FUNCTION_BLOCK FINAL Receiver IMPLEMENTS I_ReceiverNode, I_Receiver
VAR
	_iCallable		: I_Callable;
	_tag			: Tags.Tag;
	_bIsOk			: BOOL := TRUE;
END_VAR

//FB_Init is always available implicitly and it is used primarily for initialization.
//The return value is not evaluated. For a specific influence, you can also declare the
//methods explicitly and provide additional code there with the standard initialization
//code. You can evaluate the return value.
METHOD FB_Init: BOOL
VAR_INPUT
    bInitRetains: BOOL; // TRUE: the retain variables are initialized (reset warm / reset cold)
    bInCopyCode: BOOL;  // TRUE: the instance will be copied to the copy code afterward (online change)

	iCallable	: I_Callable;
END_VAR
_iCallable := iCallable;
IF _iCallable = 0 THEN
	_bIsOk := FALSE;
	Debug.DebugMsg(THIS^, 'iReceiver = 0!');
END_IF
END_METHOD

PROPERTY INTERNAL IsOk : BOOL
GET
IsOk := _bIsOk;
END_GET
END_PROPERTY

METHOD Pair : Results.Result
VAR_INPUT
	iSignal		: I_Signal;
END_VAR
IF iSignal <> 0 THEN
	Pair := iSignal.Pair(THIS^);
ELSE
	Pair := Results.Error;
END_IF
END_METHOD

METHOD INTERNAL Receive
VAR_INPUT
	iArg			: I_Arg;
END_VAR
_iCallable.Call(iArg);
END_METHOD

PROPERTY Tag : Tags.I_Tag
GET
Tag := _tag;
END_GET
END_PROPERTY

METHOD Unpair : Results.Result
VAR_INPUT
	iSignal		: I_Signal;
END_VAR
IF iSignal <> 0 THEN
	Unpair := iSignal.Unpair(THIS^);
ELSE
	Unpair := Results.Error;
END_IF
END_METHOD

END_FUNCTION_BLOCK

(* stored: Version 1.1.0.1
   POU Receiver: Id {257bc56d-d4ab-4dfa-8333-731f29b2e514}, SpecialFunc None
   Method FB_init: Id {951a002b-ff7a-48cf-b743-6a05c2c3370f}
   Property IsOk: Id {4a36423a-d62a-4434-aa29-147d4a2a72c0}
   Get Get: Id {9181fb34-27f0-4f1d-8d52-cbee4d6fcb65}
   Method Pair: Id {27407187-acff-4901-8f63-f09886ed298e}
   Method Receive: Id {34f6591a-4c68-42fe-83cd-983703da5774}
   Property Tag: Id {93b0a7a7-1505-4fb2-9b7a-4f06daa0687d}
   Get Get: Id {05560be5-36b7-415d-aeaa-e1a122c5c12d}
   Method Unpair: Id {3df2d2d8-e509-442b-918c-ed9c88636eda} *)
